(* Logix 5000 project; controller Topping_Comorfords vendor 1 type 14 code 222 rev 33.11; software revision 33.00 *)

TASK MainTask (continuous, watchdog 500 ms) : MainProgram
TASK SafetyTask (periodic, rate 20 ms, priority 10, watchdog 20 ms, safety) : SafetyProgram

MODULES
   Local : vendor 1 type 14 code 222 (5069 0, rev 33.11)
      WTU_C1_C2 : vendor 1 type 0 code 23 (Ethernet 192.168.2.12, rev 1.1)   // water tempering unit PLC
      PF525_FeedingPump_Color_2 : PowerFlex 525-EENET (Ethernet 192.168.2.18, rev 5.2, Output RPI 20 ms)   // 0.75 kW
      PF525_FeedingPump_Color_3 : PowerFlex 525-EENET (Ethernet 192.168.2.19, rev 5.2, Output RPI 20 ms)   // 0.75 kW
      PF525_FeedingPump_NO_Color : PowerFlex 525-EENET (Ethernet 192.168.2.20, rev 5.2, Output RPI 20 ms)   // 0.75 kW
      PF525_Stirrer : PowerFlex 525-EENET (Ethernet 192.168.2.14, rev 5.2, Output RPI 20 ms)   // 4 kW
      PF525_Feeding_Pump : PowerFlex 525-EENET (Ethernet 192.168.2.15, rev 5.2, Output RPI 20 ms)   // 0.75 kW
      PF525_CIP_Pump : PowerFlex 525-EENET (Ethernet 192.168.2.16, rev 5.2, Output RPI 20 ms)   // 0.75 kW
      PF525_FeedingPump_Color_1 : PowerFlex 525-EENET (Ethernet 192.168.2.17, rev 5.2, Output RPI 20 ms)   // 0.75 kW
      X_Axis : 2198-H008-ERS2 (Ethernet 192.168.2.26, rev 7.1, AMotionDiagnostics RPI 1 ms, CSafety_Output RPI 20 ms, DSafety_Input RPI 10 ms)
      Convayer : 2198-H008-ERS2 (Ethernet 192.168.2.29, rev 7.1, AMotionDiagnostics RPI 1 ms, CSafety_Output RPI 20 ms, DSafety_Input RPI 10 ms)
      Manifold_Color_1 : 2198-H008-ERS2 (Ethernet 192.168.2.22, rev 7.1, AMotionDiagnostics RPI 1 ms, CSafety_Output RPI 20 ms, DSafety_Input RPI 10 ms)
      Manifold_Color_2 : 2198-H008-ERS2 (Ethernet 192.168.2.23, rev 7.1, AMotionDiagnostics RPI 1 ms, CSafety_Output RPI 20 ms, DSafety_Input RPI 10 ms)
      Manifold_Color_3 : 2198-H008-ERS2 (Ethernet 192.168.2.24, rev 7.1, AMotionDiagnostics RPI 1 ms, CSafety_Output RPI 20 ms, DSafety_Input RPI 10 ms)
      Manifold_NO_Color : 2198-H008-ERS2 (Ethernet 192.168.2.25, rev 7.1, AMotionDiagnostics RPI 1 ms, CSafety_Output RPI 20 ms, DSafety_Input RPI 10 ms)
      Y_Axis : 2198-H008-ERS2 (Ethernet 192.168.2.27, rev 7.1, AMotionDiagnostics RPI 1 ms, CSafety_Output RPI 20 ms, DSafety_Input RPI 10 ms)
      Z_Axis : 2198-H008-ERS2 (Ethernet 192.168.2.28, rev 7.1, AMotionDiagnostics RPI 1 ms, CSafety_Output RPI 20 ms, DSafety_Input RPI 10 ms)
      U3_MCC1_IO : 1734-AENTR (Ethernet 192.168.2.13, rev 6.1, Output RPI 20 ms)
         U3_MCC1_DIG_In_1 : 1734-IB8 (PointIO 3, rev 3.1)
         U3_MCC1_DIG_In_2 : 1734-IB8 (PointIO 4, rev 3.1)
         U3_MCC1_DIG_In_3 : 1734-IB8 (PointIO 5, rev 3.1)
         U3_MCC1_DIG_In_4 : 1734-IB8 (PointIO 6, rev 3.1)
         U3_MCC1_ANA_In_1 : vendor 1 type 115 code 210 (PointIO 7, rev 3.1, Input RPI 80 ms)
         U3_MCC1_DIG_Out_1 : vendor 1 type 7 code 231 (PointIO 8, rev 3.1)
         U3_MCC1_DIG_Out_2 : 1734-OB8 (PointIO 9, rev 3.1)
         U3_MCC1_DIG_Out_3 : 1734-OB8 (PointIO 10, rev 3.1)
         U3_MCC1_DIG_Out_4 : 1734-OB8 (PointIO 11, rev 3.1)
         U3_MCC1_DIG_Out_5 : 1734-OB8 (PointIO 12, rev 3.1)
         U3_MCC1_ANA_Out_1 : 1734-OE2C (PointIO 13, rev 3.1, Output RPI 80 ms)
         U3_MCC1_ANA_Out_2 : 1734-OE2C (PointIO 14, rev 3.1, Output RPI 80 ms)
         U3_MCC1_Safety_DIG_In_1 : vendor 1 type 35 code 15 (PointIO 1, rev 2.1, Input RPI 10 ms, Output RPI 20 ms)
         U3_MCC1_Safety_DIG_Out_1 : vendor 1 type 35 code 16 (PointIO 2, rev 2.1, Input RPI 10 ms, Output RPI 20 ms)
      U6_MCC1_IO : 1734-AENTR (Ethernet 192.168.2.21, rev 6.1, Output RPI 20 ms)
         U6_MCC1_DIG_In_1 : 1734-IB8 (PointIO 3, rev 3.1)
         U6_MCC1_DIG_In_2 : 1734-IB8 (PointIO 4, rev 3.1)
         U6_MCC1_DIG_In_3 : 1734-IB8 (PointIO 5, rev 3.1)
         U6_MCC1_ANA_In_1 : vendor 1 type 115 code 210 (PointIO 6, rev 3.1, Input RPI 80 ms)
         U6_MCC1_ANA_In_2 : 1734-IE4C (PointIO 7, rev 3.1, Input RPI 80 ms)
         U6_MCC1_DIG_Out_1 : vendor 1 type 7 code 231 (PointIO 8, rev 3.1)
         U6_MCC1_DIG_Out_2 : vendor 1 type 7 code 231 (PointIO 9, rev 3.1)
         U6_MCC1_DIG_Out_3 : vendor 1 type 7 code 231 (PointIO 10, rev 3.1)
         U6_MCC1_DIG_Out_4 : vendor 1 type 7 code 231 (PointIO 11, rev 3.1)
         U6_MCC1_ANA_Out_1 : 1734-OE2C (PointIO 12, rev 3.1, Output RPI 80 ms)
         U6_MCC1_ANA_Out_2 : 1734-OE2C (PointIO 13, rev 3.1, Output RPI 80 ms)
         U6_MCC1_Safety_DIG_Out_1 : vendor 1 type 35 code 16 (PointIO 2, rev 2.1, Output RPI 20 ms, Input RPI 10 ms)
         U6_MCC1_Safety_DIG_In_1 : vendor 1 type 35 code 15 (PointIO 1, rev 2.1, Input RPI 10 ms, Output RPI 20 ms)
END_MODULES

VAR_GLOBAL   (* controller tags *)
   IA_2_1_PT01 : ALIAS FOR U3_MCC1_IO:7:I.Ch1Data;   // Pressure feeding pump 1
   IA_3_1_LT01 : ALIAS FOR U3_MCC1_IO:7:I.Ch0Data;   // Level buffertank
   IA_3_2_LT01 : ALIAS FOR U3_MCC1_IO:7:I.Ch2Data;   // Level buffertank
   IA_3_3_LT01 : ALIAS FOR U3_MCC1_IO:7:I.Ch3Data;   // Level buffertank
   IA_3_4_LT01 : ALIAS FOR U3_MCC1_IO:7:I.Ch4Data;   // Level buffertank
   IA_6_1_PT01 : ALIAS FOR U6_MCC1_IO:6:I.Ch1Data;   // Pressure manifold Color 1
   IA_6_1_PT02 : ALIAS FOR U6_MCC1_IO:6:I.Ch3Data;   // Pressure manifold Color 2
   IA_6_1_PT03 : ALIAS FOR U6_MCC1_IO:6:I.Ch5Data;   // Pressure manifold Color 3
   IA_6_1_PT04 : ALIAS FOR U6_MCC1_IO:6:I.Ch7Data;   // Pressure manifold No Color
   IA_6_1_TT01 : ALIAS FOR U6_MCC1_IO:6:I.Ch0Data;   // Temperature manifold Color 1
   IA_6_1_TT02 : ALIAS FOR U6_MCC1_IO:6:I.Ch2Data;   // Temperature manifold Color 2
   IA_6_1_TT03 : ALIAS FOR U6_MCC1_IO:6:I.Ch4Data;   // Temperature manifold Color 3
   IA_6_1_TT04 : ALIAS FOR U6_MCC1_IO:6:I.Ch6Data;   // Temperature manifold No Color
   ID_2_1_LS01 : ALIAS FOR U3_MCC1_IO:4:I.5;   // Level switch feeding pump 1
   ID_2_1_OL_CIP : ALIAS FOR U3_MCC1_IO:4:I.6;   // Thermal overload CIP pump
   ID_2_1_OL_M02 : ALIAS FOR U3_MCC1_IO:4:I.4;   // Thermal overload feeding pump 1
   ID_3_1_GS01_1 : ALIAS FOR U3_MCC1_IO:4:I.1;   // Guard switch 1.1
   ID_3_1_GS01_2 : ALIAS FOR U3_MCC1_IO:4:I.2;   // Guard switch 1.2
   ID_3_1_GS01_3 : ALIAS FOR U3_MCC1_IO:4:I.3;   // Guard switch 1.3
   ID_3_1_OL_CAB5A : ALIAS FOR U3_MCC1_IO:5:I.3;   // Thermal overload Cabinet 5A
   ID_3_1_OL_FAN : ALIAS FOR U3_MCC1_IO:3:I.0;   // Thermal overload Fan / Service socket
   ID_3_1_OL_M01 : ALIAS FOR U3_MCC1_IO:4:I.0;   // Thermal overload strirrer
   ID_3_1_PS01 : ALIAS FOR U3_MCC1_IO:3:I.1;   // Air pressure available
   ID_3_2_OL_FAN : ALIAS FOR U3_MCC1_IO:3:I.2;   // Thermal overload Fan / Service socket
   ID_3_2_OL_M01 : ALIAS FOR U3_MCC1_IO:5:I.0;   // Thermal overload Color injection pump
   ID_3_2_OL_M02 : ALIAS FOR U3_MCC1_IO:5:I.4;   // Thermal overload feeding pump Color 1
   ID_3_2_XY01_C : ALIAS FOR U3_MCC1_IO:6:I.1;   // Feedback valve 03_02_CV01 closed
   ID_3_2_XY01_O : ALIAS FOR U3_MCC1_IO:6:I.0;   // Feedback valve 03_02_CV01 open
   ID_3_3_OL_M01 : ALIAS FOR U3_MCC1_IO:5:I.1;   // Thermal overload Color injection pump
   ID_3_3_OL_M02 : ALIAS FOR U3_MCC1_IO:5:I.5;   // Thermal overload feeding pump Color 2
   ID_3_3_XY01_C : ALIAS FOR U3_MCC1_IO:6:I.3;   // Feedback valve 03_03_CV01 closed
   ID_3_3_XY01_O : ALIAS FOR U3_MCC1_IO:6:I.2;   // Feedback valve 03_03_CV01 open
   ID_3_4_OL_M01 : ALIAS FOR U3_MCC1_IO:5:I.2;   // Thermal overload Color injection pump
   ID_3_4_OL_M02 : ALIAS FOR U3_MCC1_IO:5:I.6;   // Thermal overload feeding pump Color 3
   ID_3_4_XY01_C : ALIAS FOR U3_MCC1_IO:6:I.5;   // Feedback valve 03_04_CV01 closed
   ID_3_4_XY01_O : ALIAS FOR U3_MCC1_IO:6:I.4;   // Feedback valve 03_04_CV01 open
   ID_3_5_OL_M01 : ALIAS FOR U3_MCC1_IO:5:I.7;   // Thermal overload feeding pump no Color
   ID_3_5_XY01_C : ALIAS FOR U3_MCC1_IO:6:I.7;   // Feedback valve 03_05_CV01 closed
   ID_3_5_XY01_O : ALIAS FOR U3_MCC1_IO:6:I.6;   // Feedback valve 03_05_CV01 open
   ID_6_1_GS01_1 : ALIAS FOR U6_MCC1_IO:4:I.0;   // Guard switch 1.1
   ID_6_1_GS01_2 : ALIAS FOR U6_MCC1_IO:4:I.1;   // Guard switch 1.2
   ID_6_1_GS01_3 : ALIAS FOR U6_MCC1_IO:4:I.2;   // Guard switch 1.3
   ID_6_1_GS02_1 : ALIAS FOR U6_MCC1_IO:4:I.3;   // Guard switch 2.1
   ID_6_1_GS02_2 : ALIAS FOR U6_MCC1_IO:4:I.4;   // Guard switch 2.2
   ID_6_1_GS02_3 : ALIAS FOR U6_MCC1_IO:4:I.5;   // Guard switch 2.3
   ID_6_1_GS03_1 : ALIAS FOR U6_MCC1_IO:5:I.0;   // Guard switch 3.1
   ID_6_1_GS03_2 : ALIAS FOR U6_MCC1_IO:5:I.1;   // Guard switch 3.2
   ID_6_1_GS03_3 : ALIAS FOR U6_MCC1_IO:5:I.2;   // Guard switch 3.3
   ID_6_1_GS04_1 : ALIAS FOR U6_MCC1_IO:5:I.3;   // Guard switch 4.1
   ID_6_1_GS04_2 : ALIAS FOR U6_MCC1_IO:5:I.4;   // Guard switch 4.2
   ID_6_1_GS04_3 : ALIAS FOR U6_MCC1_IO:5:I.5;   // Guard switch 4.3
   ID_6_1_OL_FAN : ALIAS FOR U6_MCC1_IO:3:I.0;   // Thermal overload Fan / Service socket
   ID_6_1_OL_M01 : ALIAS FOR U6_MCC1_IO:3:I.4;   // Thermal overload Power servo's
   ID_6_1_PS01 : ALIAS FOR U6_MCC1_IO:3:I.1;   // Air pressure available
   OA_3_2_M01 : ALIAS FOR U3_MCC1_IO:13:O.Ch0Data;   // Setpoint color pump
   OA_3_3_M01 : ALIAS FOR U3_MCC1_IO:13:O.Ch1Data;   // Setpoint color pump
   OA_3_4_M01 : ALIAS FOR U3_MCC1_IO:14:O.Ch0Data;   // Setpoint color pump
   OA_6_1_CV01 : ALIAS FOR U6_MCC1_IO:12:O.Ch0Data;   // Pressure valve manifold Color 1
   OA_6_1_CV02 : ALIAS FOR U6_MCC1_IO:12:O.Ch1Data;   // Pressure valve manifold Color 2
   OA_6_1_CV03 : ALIAS FOR U6_MCC1_IO:13:O.Ch0Data;   // Pressure valve manifold Color 3
   OA_6_1_CV04 : ALIAS FOR U6_MCC1_IO:13:O.Ch1Data;   // Pressure valve manifold No Color
   OD_3_1_CV01 : ALIAS FOR U3_MCC1_IO:10:O.0;   // Drain after tank
   OD_3_1_CV02 : ALIAS FOR U3_MCC1_IO:10:O.1;   // Bypass CIP before
   OD_3_1_CV03 : ALIAS FOR U3_MCC1_IO:10:O.2;   // Drain before CIP pump
   OD_3_1_CV04 : ALIAS FOR U3_MCC1_IO:10:O.3;   // Bypass CIP after
   OD_3_1_CV05 : ALIAS FOR U3_MCC1_IO:10:O.4;   // Product return
   OD_3_1_CV06 : ALIAS FOR U3_MCC1_IO:10:O.5;   // Drain before tank
   OD_3_1_CV07 : ALIAS FOR U3_MCC1_IO:10:O.6;   // Return tank
   OD_3_1_CV08 : ALIAS FOR U3_MCC1_IO:10:O.7;   // Sprinkler
   OD_3_1_CV09 : ALIAS FOR U3_MCC1_IO:11:O.0;   // Return icing tank
   OD_3_1_CV10 : ALIAS FOR U3_MCC1_IO:11:O.1;   // Return cream tank
   OD_3_1_CV11 : ALIAS FOR U3_MCC1_IO:11:O.2;   // Hot water inlet
   OD_3_1_CV12 : ALIAS FOR U3_MCC1_IO:11:O.3;   // Cold water inlet
   OD_3_1_CV13 : ALIAS FOR U3_MCC1_IO:11:O.4;   // From Cream tank
   OD_3_1_CV14 : ALIAS FOR U3_MCC1_IO:11:O.5;   // From icing tank
   OD_3_1_CV15 : ALIAS FOR U3_MCC1_IO:11:O.6;   // Spare
   OD_3_1_CV16 : ALIAS FOR U3_MCC1_IO:11:O.7;   // Spare
   OD_3_1_GS01 : ALIAS FOR U3_MCC1_IO:9:O.0;   // Guard switch 1 lock
   OD_3_1_SLBZ : ALIAS FOR U3_MCC1_IO:8:O.3;   // Signal column BUZZER
   OD_3_1_SLGN : ALIAS FOR U3_MCC1_IO:8:O.0;   // Signal column GN
   OD_3_1_SLRD : ALIAS FOR U3_MCC1_IO:8:O.2;   // Signal column RD
   OD_3_1_SLYE : ALIAS FOR U3_MCC1_IO:8:O.1;   // Signal column YE
   OD_3_2_CV01 : ALIAS FOR U3_MCC1_IO:12:O.0;   // Drain color 1 tank
   OD_3_2_CV02 : ALIAS FOR U3_MCC1_IO:12:O.1;   // To color 1
   OD_3_2_M01 : ALIAS FOR U3_MCC1_IO:9:O.1;   // Enable color pump
   OD_3_3_CV01 : ALIAS FOR U3_MCC1_IO:12:O.2;   // Drain color 2 tank
   OD_3_3_CV02 : ALIAS FOR U3_MCC1_IO:12:O.3;   // To color 2
   OD_3_3_M01 : ALIAS FOR U3_MCC1_IO:9:O.2;   // Enable color pump
   OD_3_4_CV01 : ALIAS FOR U3_MCC1_IO:12:O.4;   // Drain color 3 tank
   OD_3_4_CV02 : ALIAS FOR U3_MCC1_IO:12:O.5;   // To color 3
   OD_3_4_M01 : ALIAS FOR U3_MCC1_IO:9:O.3;   // Enable color pump
   OD_3_5_CV01 : ALIAS FOR U3_MCC1_IO:12:O.6;   // Bypass colors
   OD_3_5_CV02 : ALIAS FOR U3_MCC1_IO:12:O.7;   // Spare
   OD_6_1_CV01 : ALIAS FOR U6_MCC1_IO:10:O.0;   // Valve before manifold Color 1
   OD_6_1_CV02 : ALIAS FOR U6_MCC1_IO:10:O.1;   // Valve before manifold Color 2
   OD_6_1_CV03 : ALIAS FOR U6_MCC1_IO:10:O.2;   // Valve before manifold Color 3
   OD_6_1_CV04 : ALIAS FOR U6_MCC1_IO:10:O.3;   // Valve before manifold No Color
   OD_6_1_GS01 : ALIAS FOR U6_MCC1_IO:9:O.0;   // Guard switch 1 lock
   OD_6_1_GS02 : ALIAS FOR U6_MCC1_IO:9:O.1;   // Guard switch 2 lock
   OD_6_1_GS03 : ALIAS FOR U6_MCC1_IO:9:O.2;   // Guard switch 3 lock
   OD_6_1_GS04 : ALIAS FOR U6_MCC1_IO:9:O.3;   // Guard switch 4 lock
   OD_6_1_SLBZ : ALIAS FOR U6_MCC1_IO:8:O.3;   // Signal column BUZZER
   OD_6_1_SLGN : ALIAS FOR U6_MCC1_IO:8:O.0;   // Signal column GN
   OD_6_1_SLRD : ALIAS FOR U6_MCC1_IO:8:O.2;   // Signal column RD
   OD_6_1_SLYE : ALIAS FOR U6_MCC1_IO:8:O.1;   // Signal column YE
END_VAR

PROGRAM MainProgram   (* main routine MainRoutine *)

ROUTINE MainRoutine   (* ladder *)
END_ROUTINE
END_PROGRAM

PROGRAM SafetyProgram   (* main routine MainRoutine, safety *)

ROUTINE MainRoutine   (* ladder *)
END_ROUTINE
END_PROGRAM
